// TwinCAT 3 PLC project plc_qrixs_vac
// ProgramVersion: 3.1.4022.7
// libraries:
//   LCLS General, * (SLAC)
//   LCLS Vacuum, * (SLAC - LCLS)
//   PMPS, * (SLAC - LCLS)
//   Tc2_Standard, * (Beckhoff Automation GmbH)
//   Tc2_System, * (Beckhoff Automation GmbH)
//   Tc3_Module, * (Beckhoff Automation GmbH)
// project tree:
//   GVLs/ GVL_Devices.TcGVL, GVL_PMPS.TcGVL, GVL_Variables.TcGVL
//   / PlcTask.TcTTO
//   POUs/ MAIN.TcPOU
// real-time tasks:
//   TASK PlcTask: cycle T#10ms, priority 20, ADS port 350
// I/O:
//   DEVICE Device 1 (EtherCAT), AmsNetId 5.85.195.62.2.1
//     qRIXS_PLC_E0_EK1200 [EK1200-5000 EtherCAT Power supply (2A E-Bus)]
//       qRIXS_PLC_E1_EL1004 [EL1004 4Ch. Dig. Input 24V, 3ms]
//       qRIXS_PLC_E2_EL2794 [EL2794 4Ch. Dig. Output 24V AC/DC, 2A, short-circuit-proof]
//       qRIXS_PLC_E3_EL3064 [EL3064 4Ch. Ana. Input 0-10V]
//       qRIXS_PLC_E4_EK1122 [EK1122 2 port EtherCAT junction]
//         qRIXS_PNL1_E0_EK1100 [EK1100 EtherCAT Coupler (2A E-Bus)]
//           qRIXS_PNL1_E1_EL1004 [EL1004 4Ch. Dig. Input 24V, 3ms]
//           qRIXS_PNL1_E2_EL1004 [EL1004 4Ch. Dig. Input 24V, 3ms]
//           qRIXS_PNL1_E3_EL2004 [EL2004 4Ch. Dig. Output 24V, 0.5A]
//           qRIXS_PNL1_E4_EL2624 [EL2624 4Ch. Relay Output, NO (125V AC / 30V DC)]
//           qRIXS_PNL1_E5_EL3174-0002 [EL3174-0002 4Ch. Ana. Input +/-10V, +/-20mA 16 Bit, Isolated Channels]
//           qRIXS_PNL1_E6_EL3174-0002 [EL3174-0002 4Ch. Ana. Input +/-10V, +/-20mA 16 Bit, Isolated Channels]
//           qRIXS_PNL1_E7_EL9505 [EL9505 Power supply terminal 5V]
//           qRIXS_PNL1_E8_EL1124 [EL1124 4Ch. Dig. Input 5V, 10µs, Sensor Power]
//           qRIXS_PNL1_E9_EL9410 [EL9410 E-Bus Power Supplier  (Diagnostics)]
//           qRIXS_PNL1_E10_EK1110 [EK1110 EtherCAT extension]
// variable links:
//   plc_qrixs_vac/plc_qrixs_vac Instance <-> Device 1 (EtherCAT)/qRIXS_PLC_E0_EK1200/qRIXS_PLC_E1_EL1004
//     PlcTask Inputs/GVL_Devices.qRIXS_DET_PIP_01.i_xSP_DI <-> Channel 2/Input
//     PlcTask Inputs/GVL_Devices.qRIXS_OPT_PIP_01.i_xSP_DI <-> Channel 1/Input
//   plc_qrixs_vac/plc_qrixs_vac Instance <-> Device 1 (EtherCAT)/qRIXS_PLC_E0_EK1200/qRIXS_PLC_E2_EL2794
//     PlcTask Outputs/GVL_Devices.qRIXS_DET_PIP_01.q_xHVEna_DO <-> Channel 2/Output
//     PlcTask Outputs/GVL_Devices.qRIXS_OPT_PIP_01.q_xHVEna_DO <-> Channel 1/Output
//   plc_qrixs_vac/plc_qrixs_vac Instance <-> Device 1 (EtherCAT)/qRIXS_PLC_E0_EK1200/qRIXS_PLC_E3_EL3064
//     PlcTask Inputs/GVL_Devices.qRIXS_DET_PIP_01.i_iPRESS <-> AI Standard Channel 2/Value
//     PlcTask Inputs/GVL_Devices.qRIXS_OPT_PIP_01.i_iPRESS <-> AI Standard Channel 1/Value
//   plc_qrixs_vac/plc_qrixs_vac Instance <-> Device 1 (EtherCAT)/qRIXS_PLC_E0_EK1200/qRIXS_PLC_E4_EK1122/qRIXS_PNL1_E0_EK1100/qRIXS_PNL1_E1_EL1004
//     PlcTask Inputs/GVL_Devices.qRIXS_BLW_VRC_01.i_xClsLS <-> Channel 4/Input
//     PlcTask Inputs/GVL_Devices.qRIXS_BLW_VRC_01.i_xOpnLS <-> Channel 3/Input
//     PlcTask Inputs/GVL_Devices.qRIXS_OPT_VGC_01.i_xClsLS <-> Channel 2/Input
//     PlcTask Inputs/GVL_Devices.qRIXS_OPT_VGC_01.i_xOpnLS <-> Channel 1/Input
//   plc_qrixs_vac/plc_qrixs_vac Instance <-> Device 1 (EtherCAT)/qRIXS_PLC_E0_EK1200/qRIXS_PLC_E4_EK1122/qRIXS_PNL1_E0_EK1100/qRIXS_PNL1_E2_EL1004
//     PlcTask Inputs/GVL_Devices.qRIXS_DET_VRC_01.i_xClsLS <-> Channel 2/Input
//     PlcTask Inputs/GVL_Devices.qRIXS_DET_VRC_01.i_xOpnLS <-> Channel 1/Input
//   plc_qrixs_vac/plc_qrixs_vac Instance <-> Device 1 (EtherCAT)/qRIXS_PLC_E0_EK1200/qRIXS_PLC_E4_EK1122/qRIXS_PNL1_E0_EK1100/qRIXS_PNL1_E3_EL2004
//     PlcTask Outputs/GVL_Devices.qRIXS_BLW_VRC_01.q_xOPN_DO <-> Channel 2/Output
//     PlcTask Outputs/GVL_Devices.qRIXS_DET_VRC_01.q_xOPN_DO <-> Channel 3/Output
//     PlcTask Outputs/GVL_Devices.qRIXS_OPT_VGC_01.q_xOPN_DO <-> Channel 1/Output
//   plc_qrixs_vac/plc_qrixs_vac Instance <-> Device 1 (EtherCAT)/qRIXS_PLC_E0_EK1200/qRIXS_PLC_E4_EK1122/qRIXS_PNL1_E0_EK1100/qRIXS_PNL1_E4_EL2624
//     PlcTask Outputs/GVL_Devices.qRIXS_DET_GCC_01.q_xHV_DIS <-> Channel 2/Output
//     PlcTask Outputs/GVL_Devices.qRIXS_OPT_GCC_01.q_xHV_DIS <-> Channel 1/Output
//   plc_qrixs_vac/plc_qrixs_vac Instance <-> Device 1 (EtherCAT)/qRIXS_PLC_E0_EK1200/qRIXS_PLC_E4_EK1122/qRIXS_PNL1_E0_EK1100/qRIXS_PNL1_E5_EL3174-0002
//     PlcTask Inputs/GVL_Devices.qRIXS_BLW_GFR_01.i_iPRESS_R <-> AI Standard Channel 3/Value
//     PlcTask Inputs/GVL_Devices.qRIXS_DET_GPI_01.i_iPRESS_R <-> AI Standard Channel 2/Value
//     PlcTask Inputs/GVL_Devices.qRIXS_OPT_GPI_01.i_iPRESS_R <-> AI Standard Channel 1/Value
//   plc_qrixs_vac/plc_qrixs_vac Instance <-> Device 1 (EtherCAT)/qRIXS_PLC_E0_EK1200/qRIXS_PLC_E4_EK1122/qRIXS_PNL1_E0_EK1100/qRIXS_PNL1_E6_EL3174-0002
//     PlcTask Inputs/GVL_Devices.qRIXS_DET_GCC_01.i_iPRESS_R <-> AI Standard Channel 2/Value
//     PlcTask Inputs/GVL_Devices.qRIXS_OPT_GCC_01.i_iPRESS_R <-> AI Standard Channel 1/Value
//   plc_qrixs_vac/plc_qrixs_vac Instance <-> Device 1 (EtherCAT)/qRIXS_PLC_E0_EK1200/qRIXS_PLC_E4_EK1122/qRIXS_PNL1_E0_EK1100/qRIXS_PNL1_E8_EL1124
//     PlcTask Inputs/GVL_Devices.qRIXS_DET_GCC_01.i_xDisc_Active <-> Channel 4/Input
//     PlcTask Inputs/GVL_Devices.qRIXS_DET_GCC_01.i_xHV_ON <-> Channel 3/Input
//     PlcTask Inputs/GVL_Devices.qRIXS_OPT_GCC_01.i_xDisc_Active <-> Channel 2/Input
//     PlcTask Inputs/GVL_Devices.qRIXS_OPT_GCC_01.i_xHV_ON <-> Channel 1/Input

CONFIGURATION plc_qrixs_vac
    RESOURCE PLC ON TwinCAT3
        TASK PlcTask(INTERVAL := T#10ms, PRIORITY := 20);
        PROGRAM MAIN WITH PlcTask : MAIN;
    END_RESOURCE
END_CONFIGURATION

// ---- GVLs/GVL_Devices.TcGVL
//{attribute 'qualified_only'}
VAR_GLOBAL
	(* Gamma Ion Pump *)
	{attribute 'TcLinkTo' := 	'.q_xHVEna_DO	:=	TIIB[qRIXS_PLC_E2_EL2794]^Channel 1^Output;
								 .i_iPRESS		:=	TIIB[qRIXS_PLC_E3_EL3064]^AI Standard Channel 1^Value;
								 .i_xSP_DI		:=	TIIB[qRIXS_PLC_E1_EL1004]^Channel 1^Input
	'}
	{attribute 'pytmc' := '
		pv: QRIXS:OPT:PIP:01
		io: io
	'}
	qRIXS_OPT_PIP_01: FB_PIP_Gamma;
	
	(* Gamma Ion Pump *)
	{attribute 'TcLinkTo' := 	'.q_xHVEna_DO	:=	TIIB[qRIXS_PLC_E2_EL2794]^Channel 2^Output;
								 .i_iPRESS		:=	TIIB[qRIXS_PLC_E3_EL3064]^AI Standard Channel 2^Value;
								 .i_xSP_DI		:=	TIIB[qRIXS_PLC_E1_EL1004]^Channel 2^Input
	'}
	{attribute 'pytmc' := '
		pv: QRIXS:DET:PIP:01
		io: io
	'}
	qRIXS_DET_PIP_01: FB_PIP_Gamma;	
	
	
	(* -- Normally Closed Valve with Readback -- *)
	{attribute 'TcLinkTo' := 	'.i_xOpnLS	:=	TIIB[qRIXS_PNL1_E1_EL1004]^Channel 1^Input;
								 .i_xClsLS	:=	TIIB[qRIXS_PNL1_E1_EL1004]^Channel 2^Input;
								 .q_xOPN_DO	:=	TIIB[qRIXS_PNL1_E3_EL2004]^Channel 1^Output
	'}
	{attribute 'pytmc' := '
		pv: QRIXS:OPT:VGC:01
		io: io
	'}
	qRIXS_OPT_VGC_01: FB_VGC;
		
	{attribute 'TcLinkTo' := 	'.i_xOpnLS	:=	TIIB[qRIXS_PNL1_E1_EL1004]^Channel 3^Input;
								 .i_xClsLS	:=	TIIB[qRIXS_PNL1_E1_EL1004]^Channel 4^Input;
								 .q_xOPN_DO	:=	TIIB[qRIXS_PNL1_E3_EL2004]^Channel 2^Output
	'}
	{attribute 'pytmc' := '
		pv: QRIXS:BLW:VRC:01
		io: io
	'}
	qRIXS_BLW_VRC_01: FB_VRC;
	
	{attribute 'TcLinkTo' := 	'.i_xOpnLS	:=	TIIB[qRIXS_PNL1_E2_EL1004]^Channel 1^Input;
								 .i_xClsLS	:=	TIIB[qRIXS_PNL1_E2_EL1004]^Channel 2^Input;
								 .q_xOPN_DO	:=	TIIB[qRIXS_PNL1_E3_EL2004]^Channel 3^Output
	'}
	{attribute 'pytmc' := '
		pv: QRIXS:DET:VRC:01
		io: io
	'}
	qRIXS_DET_VRC_01: FB_VRC;
	
	
	(* MKS275 - Pirani *)
	{attribute 'TcLinkTo' := 	'.i_iPRESS_R	:=	TIIB[qRIXS_PNL1_E5_EL3174-0002]^AI Standard Channel 1^Value'}
	{attribute 'pytmc' := '
		pv: QRIXS:OPT:GPI:01
		io: io
	'}
	qRIXS_OPT_GPI_01: FB_MKS275;

	{attribute 'TcLinkTo' := 	'.i_iPRESS_R	:=	TIIB[qRIXS_PNL1_E5_EL3174-0002]^AI Standard Channel 2^Value'}
	{attribute 'pytmc' := '
		pv: QRIXS:DET:GPI:01
		io: io
	'}
	qRIXS_DET_GPI_01: FB_MKS275;
	
	
	(* MKS972 - Full range guage *)
	{attribute 'TcLinkTo' := 	'.i_iPRESS_R	:=	TIIB[qRIXS_PNL1_E5_EL3174-0002]^AI Standard Channel 3^Value'}
	{attribute 'pytmc' := '
		pv: QRIXS:BLW:GFR:01
		io: io
	'}
	qRIXS_BLW_GFR_01: FB_972;
	
	
	(* MKS500 - Cold cathode gauge *)
	{attribute 'TcLinkTo' := 	'.i_iPRESS_R		:=	TIIB[qRIXS_PNL1_E6_EL3174-0002]^AI Standard Channel 1^Value;
								 .i_xHV_ON			:=	TIIB[qRIXS_PNL1_E8_EL1124]^Channel 1^Input;
								 .i_xDisc_Active	:=	TIIB[qRIXS_PNL1_E8_EL1124]^Channel 2^Input;
								 .q_xHV_DIS			:=	TIIB[qRIXS_PNL1_E4_EL2624]^Channel 1^Output
	'}
	{attribute 'pytmc' := '
		pv: QRIXS:OPT:GCC:01
		io: io
	'}
	qRIXS_OPT_GCC_01: FB_MKS500;
	
	
	{attribute 'TcLinkTo' := 	'.i_iPRESS_R		:=	TIIB[qRIXS_PNL1_E6_EL3174-0002]^AI Standard Channel 2^Value;
								 .i_xHV_ON			:=	TIIB[qRIXS_PNL1_E8_EL1124]^Channel 3^Input;
								 .i_xDisc_Active	:=	TIIB[qRIXS_PNL1_E8_EL1124]^Channel 4^Input;
								 .q_xHV_DIS			:=	TIIB[qRIXS_PNL1_E4_EL2624]^Channel 2^Output
	'}
	{attribute 'pytmc' := '
		pv: QRIXS:DET:GCC:01
		io: io
	'}
	qRIXS_DET_GCC_01: FB_MKS500;
END_VAR

// ---- GVLs/GVL_PMPS.TcGVL
{attribute 'qualified_only'}
VAR_GLOBAL
    g_FastFaultOutput1  :   FB_HardwareFFOutput;	//FFO for Upstream Components
	g_fbArbiter1: FB_Arbiter(1);
END_VAR

// ---- GVLs/GVL_Variables.TcGVL
{attribute 'qualified_only'}
VAR_GLOBAL
	{attribute 'pytmc' := '
		pv: PLC:QRIXS:VAC:OVRDON
		io: io
	'}
	xSystemOverrideMode_qRIXS	: BOOL := FALSE; (* Global system override for the qRIXS Vacuum System EBD*)

	// io_fbFFHWO: FB_FFHWO;
	
END_VAR

// ---- POUs/MAIN.TcPOU
PROGRAM MAIN
VAR
	xExtILK_OK_OPT : BOOL := True;
	xExtILK_OK_BLW : BOOL;
	xExtILK_OK_DET : BOOL;
	iPressTorrerance : REAL := 1.0; // Torr
	stUSG_dummy : ST_VG;
END_VAR


(* Gamma Ion Pump *)
	qRIXS_OPT_PIP_01(i_stGauge:=qRIXS_OPT_GCC_01.IG, i_xOverrideMode:= GVL_Variables.xSystemOverrideMode_qRIXS);
	qRIXS_DET_PIP_01(i_stGauge:=qRIXS_DET_GCC_01.IG, i_xOverrideMode:= GVL_Variables.xSystemOverrideMode_qRIXS);

(* Pirani MKS 275 Gauges *)
	qRIXS_OPT_GPI_01(PG=>);	
	qRIXS_DET_GPI_01(PG=>);

(* Full Range Gauges *)
	qRIXS_BLW_GFR_01(PG=>);

(* Cold Cathode Gauges *)
	qRIXS_OPT_GCC_01(PG:=qRIXS_OPT_GPI_01.PG, IG=>, bEP:=FALSE);
	qRIXS_DET_GCC_01(PG:=qRIXS_DET_GPI_01.PG, IG=>, bEP:=FALSE);
	
(* Normally Closed Vate Valve *)
//(*
	stUSG_dummy := qRIXS_OPT_GCC_01.IG;
	qRIXS_OPT_VGC_01(
		i_stUSG := stUSG_dummy,
		i_stDSG := qRIXS_OPT_GCC_01.IG,
		i_xExt_OK := xExtILK_OK_OPT,
		i_xOverrideMode:=GVL_Variables.xSystemOverrideMode_qRIXS,
		io_fbFFHWO := GVL_PMPS.g_FastFaultOutput1,
		fbArbiter := GVL_PMPS.g_fbArbiter1,
		iq_stValve =>,
	);
// *)
// (*
	qRIXS_BLW_VRC_01(
		i_xExtILK_OK := xExtILK_OK_BLW,
		i_xOverrideMode:=GVL_Variables.xSystemOverrideMode_qRIXS,
		iq_stValve =>
	);
// *)
// (*
	qRIXS_DET_VRC_01(
		i_xExtILK_OK := xExtILK_OK_DET,
		i_xOverrideMode:=GVL_Variables.xSystemOverrideMode_qRIXS,
		iq_stValve =>,
	);
// *)


// Calc pressure Difference
xExtILK_OK_BLW := 	( qRIXS_OPT_VGC_01.iq_stValve.i_xClsLS AND qRIXS_OPT_GPI_01.PG.xPRESS_OK AND qRIXS_BLW_GFR_01.PG.xPRESS_OK AND (qRIXS_OPT_GPI_01.PG.rPRESS - qRIXS_BLW_GFR_01.PG.rPRESS) < iPressTorrerance)
					OR (qRIXS_OPT_GCC_01.IG.xPRESS_OK AND qRIXS_BLW_GFR_01.PG.xPRESS_OK AND (qRIXS_OPT_GCC_01.IG.rPRESS - qRIXS_BLW_GFR_01.PG.rPRESS) < iPressTorrerance);
xExtILK_OK_DET := 	(qRIXS_DET_GPI_01.PG.xPRESS_OK AND qRIXS_BLW_GFR_01.PG.xPRESS_OK AND (qRIXS_DET_GPI_01.PG.rPRESS - qRIXS_BLW_GFR_01.PG.rPRESS) < iPressTorrerance)
					OR (qRIXS_DET_GCC_01.IG.xPRESS_OK AND qRIXS_BLW_GFR_01.PG.xPRESS_OK AND (qRIXS_DET_GCC_01.IG.rPRESS - qRIXS_BLW_GFR_01.PG.rPRESS) < iPressTorrerance);

END_PROGRAM
